(* PLC project PLC, Beckhoff Automation GmbH TwinCAT PLC Control 3.5.13.21 *)
(* stored: creationDateTime 2024-02-17T22:43:53.6195571, modificationDateTime 2024-02-17T22:43:53.6195571 *)

PROGRAM Unit
VAR
	stopperToUp: BOOL;
	stopperToDown: BOOL;	

	stopper: Cyl;
	fwButton: PB;
	rvButton: PB;
	
	unmatchConfigLamp: LP;
END_VAR

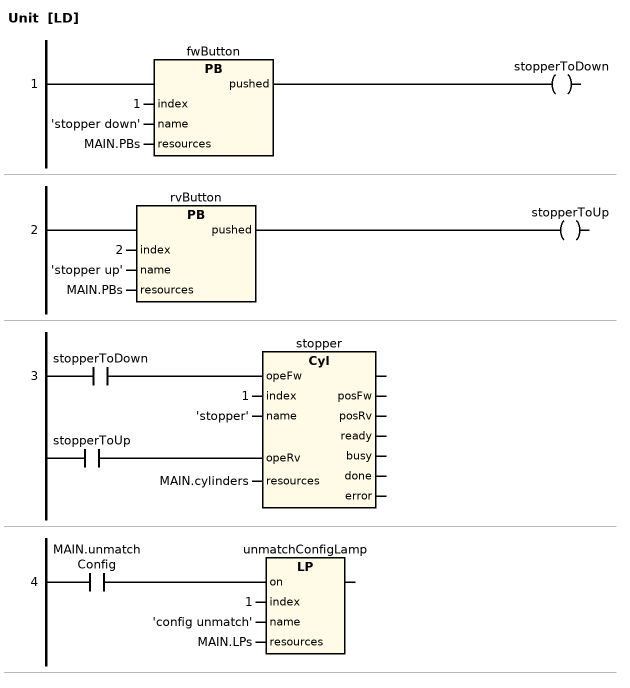
(* LD diagram, written out as Structured Text *)

fwButton(index := 1, name := 'stopper down', resources := MAIN.PBs);
stopperToDown := fwButton.pushed;

rvButton(index := 2, name := 'stopper up', resources := MAIN.PBs);
stopperToUp := rvButton.pushed;

stopper(index := 1, name := 'stopper', opeFw := stopperToDown, opeRv := stopperToUp, resources := MAIN.cylinders);

unmatchConfigLamp(index := 1, name := 'config unmatch', on := MAIN.unmatchConfig, resources := MAIN.LPs);
END_PROGRAM
